FUNCTION_BLOCK Q_Size (* Command change size ( Part 6 - F.18 ) *)
  (* Standard: ISO 11783-6; Description: The Change Size command is used to change the size of an object. Return values iso_s16 - E_NO_ERR - OK - E_OVERFLOW - buffer overflow - E_NOACT - Command not possible in current state - E_NO_INSTANCE - No VT client available *)
  (* Version 1.0, 2022-07-08, franz *)
  (* Documentation:
  The Change Size command is used to change the size of an object.
   Return values
   iso_s16
    - E_NO_ERR - OK
   - E_OVERFLOW - buffer overflow
   - E_NOACT - Command not possible in current state
   - E_NO_INSTANCE - No VT client available
  *)
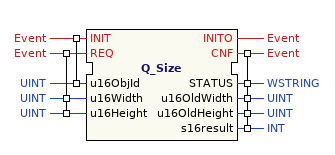
  EVENT_INPUT
    INIT WITH u16ObjId; (* Service Initialization *)
    REQ WITH u16Width, u16Height; (* Service Request *)
  END_EVENT
  EVENT_OUTPUT
    INITO; (* Initialization Confirm *)
    CNF WITH STATUS, s16result, u16OldWidth, u16OldHeight; (* Confirmation of Requested Service *)
  END_EVENT
  VAR_INPUT
    u16ObjId : UINT; (* Object ID *)
    u16Width : UINT; (* New width *)
    u16Height : UINT; (* New height *)
  END_VAR
  VAR_OUTPUT
    STATUS : WSTRING; (* Service Status *)
    u16OldWidth : UINT; (* Old width *)
    u16OldHeight : UINT; (* Old height *)
    s16result : INT; (* retval see description *)
  END_VAR
END_FUNCTION_BLOCK
